// TIA Portal V17 program export: 0 tag tables, 0 data types, 0 data blocks, 2 code blocks (in call order from the OBs), 0 instance data blocks

ORGANIZATION_BLOCK "Main"   // OB1, LAD, ProgramCycle
TITLE = "Main Program Sweep (Cycle)"
{ S7_Optimized_Access := 'TRUE' }
VERSION : 0.1
// stored: AutoNumber true, IsIECCheckEnabled false, SetENOAutomatically false
   VAR_INPUT
      Initial_Call : Bool;   // Initial call of this OB
      Remanence : Bool;   // =True, if remanent data are available
   END_VAR
BEGIN

REGION Network 1
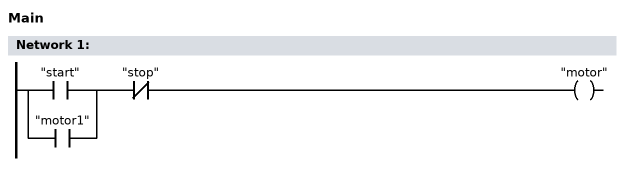
   RUNG wire#powerrail
      Contact( "start" )
      wire#w1
      I_Contact( "stop" )
      Coil( "motor" )
   END_RUNG
   RUNG wire#powerrail
      Contact( "motor1" )
   END_RUNG wire#w1
   // the same network as SCL:
   "motor" := ("start" OR "motor1") AND NOT "stop";
END_REGION
END_ORGANIZATION_BLOCK

FUNCTION_BLOCK "PID"
{ S7_Optimized_Access := 'TRUE' }
VERSION : 0.1

BEGIN

END_FUNCTION_BLOCK
